// TIA Portal V20 export
FUNCTION_BLOCK "Receive_FData"   // FB2, FBD
{ S7_Optimized_Access := 'TRUE' }
// stored: MemoryReserve 100, SetENOAutomatically false
   VAR
      TRCV_Instance { S7_SetPoint := 'True'} : TRCV;
   END_VAR
BEGIN

REGION Network 1: ACK tömb fogadása
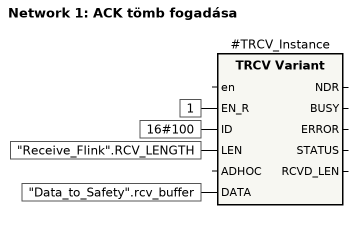
   #TRCV_Instance(EN_R := 1,   // TRCV
                  ID := 16#100,
                  LEN := "Receive_Flink".RCV_LENGTH,
                  DATA := "Data_to_Safety".rcv_buffer);
END_REGION
END_FUNCTION_BLOCK
